FUNCTION_BLOCK FB_Comau
VAR_INPUT
	
END_VAR
VAR_OUTPUT
	
END_VAR
VAR
	txData				: TxComau;	
	rxData				: RxComau;
	
	ipAddr 				: UDINT;
	remotePort 			: UINT;
	localPort 			: UINT;
	
	udpClient 			: FB_UdpClient(ipAddr, remotePort, localPort, SIZEOF(txData), ADR(txData), SIZEOF(rxData), ADR(rxData));
	
END_VAR


txData.udp_key := 32;
txData.cmnd := 0;
txData.beta := 1.0;
txData.omega := 1.0;



udpClient();

METHOD FB_init : BOOL
VAR_INPUT
	bInitRetains : BOOL; // if TRUE, the retain variables are initialized (warm start / cold start)
	bInCopyCode : BOOL;  // if TRUE, the instance afterwards gets moved into the copy code (online change)
	
	// Contructor arguments
	_ipAddr 			: UDINT;
	_remotePort 		: UINT;
	_localPort 		: UINT;
END_VAR
// Initilize parameters
ipAddr := _ipAddr;
remotePort := _remotePort;
localPort := _localPort;

// Construct FB_UdpClient
udpClient.FB_init(bInitRetains, bInCopyCode, ipAddr, remotePort, localPort, SIZEOF(txData), ADR(txData), SIZEOF(rxData), ADR(rxData));
END_METHOD

END_FUNCTION_BLOCK

(* stored: Version 1.1.0.1, ProductVersion 3.1.4020.12
   POU FB_Comau: Id {d2f3bbdf-53d6-48ce-8687-0c01a6900a56}, SpecialFunc None
   Method FB_init: Id {e628e4d7-1328-4556-8ad8-21329793d760} *)
